// TIA Portal V17 export
// export: Created 2023-03-06T02:05:17.4655163Z, ExportSetting WithDefaults, DisplayName Totally Integrated Automation Portal, DisplayVersion V17 Update 4, DisplayName TIA Portal Openness, DisplayVersion V17 Update 4, DisplayName TIA Portal Version Control Interface, DisplayVersion V17, DisplayName STEP 7 Professional, DisplayVersion V17 Update 4, DisplayName STEP 7 Safety, DisplayVersion V17, DisplayName WinCC Professional, DisplayVersion V17 Update 4
FUNCTION "AssetSt" : Void   // FC122, LAD
{ S7_Optimized_Access := 'TRUE' }
VERSION : 0.1
// stored: AutoNumber false, IsIECCheckEnabled false, SetENOAutomatically false, UDAEnableTagReadback false
BEGIN

REGION Network 1: Asset Status Battery Bank 1
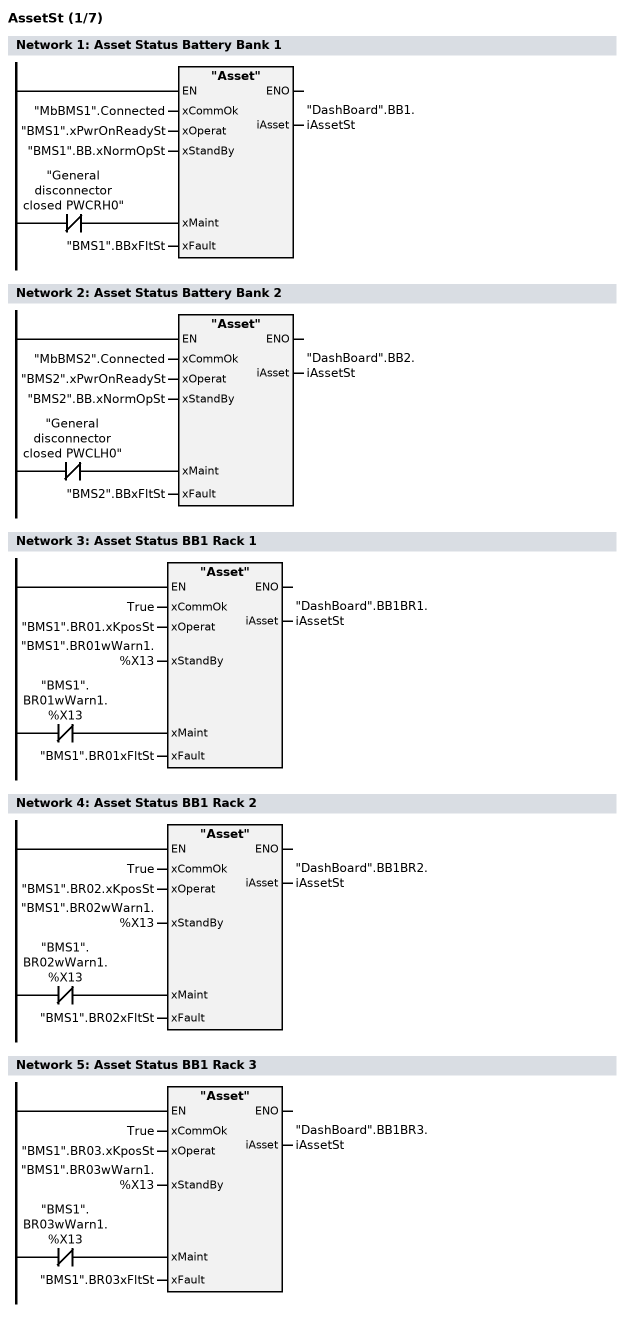
   RUNG wire#powerrail
      "Asset"(xMaint := wire#w1, xCommOk := "MbBMS1".Connected, xOperat := "BMS1".xPwrOnReadySt, xStandBy := "BMS1".BB.xNormOpSt, xFault := "BMS1".BBxFltSt, iAsset => "DashBoard".BB1.iAssetSt)
   END_RUNG
   RUNG wire#powerrail
      I_Contact( "General disconnector closed PWCRH0" )
   END_RUNG wire#w1
   // the same network as SCL:
   "Asset"(xCommOk := "MbBMS1".Connected,
           xOperat := "BMS1".xPwrOnReadySt,
           xStandBy := "BMS1".BB.xNormOpSt,
           xMaint := NOT "General disconnector closed PWCRH0",
           xFault := "BMS1".BBxFltSt,
           iAsset => "DashBoard".BB1.iAssetSt);
END_REGION

REGION Network 2: Asset Status Battery Bank 2
   RUNG wire#powerrail
      "Asset"(xMaint := wire#w1, xCommOk := "MbBMS2".Connected, xOperat := "BMS2".xPwrOnReadySt, xStandBy := "BMS2".BB.xNormOpSt, xFault := "BMS2".BBxFltSt, iAsset => "DashBoard".BB2.iAssetSt)
   END_RUNG
   RUNG wire#powerrail
      I_Contact( "General disconnector closed PWCLH0" )
   END_RUNG wire#w1
   // the same network as SCL:
   "Asset"(xCommOk := "MbBMS2".Connected,
           xOperat := "BMS2".xPwrOnReadySt,
           xStandBy := "BMS2".BB.xNormOpSt,
           xMaint := NOT "General disconnector closed PWCLH0",
           xFault := "BMS2".BBxFltSt,
           iAsset => "DashBoard".BB2.iAssetSt);
END_REGION

REGION Network 3: Asset Status BB1 Rack 1
   RUNG wire#powerrail
      "Asset"(xMaint := wire#w1, xCommOk := True, xOperat := "BMS1".BR01.xKposSt, xStandBy := "BMS1".BR01wWarn1.%X13, xFault := "BMS1".BR01xFltSt, iAsset => "DashBoard".BB1BR1.iAssetSt)
   END_RUNG
   RUNG wire#powerrail
      I_Contact( "BMS1".BR01wWarn1.%X13 )
   END_RUNG wire#w1
   // the same network as SCL:
   "Asset"(xCommOk := True,
           xOperat := "BMS1".BR01.xKposSt,
           xStandBy := "BMS1".BR01wWarn1.%X13,
           xMaint := NOT "BMS1".BR01wWarn1.%X13,
           xFault := "BMS1".BR01xFltSt,
           iAsset => "DashBoard".BB1BR1.iAssetSt);
END_REGION

REGION Network 4: Asset Status BB1 Rack 2
   RUNG wire#powerrail
      "Asset"(xMaint := wire#w1, xCommOk := True, xOperat := "BMS1".BR02.xKposSt, xStandBy := "BMS1".BR02wWarn1.%X13, xFault := "BMS1".BR02xFltSt, iAsset => "DashBoard".BB1BR2.iAssetSt)
   END_RUNG
   RUNG wire#powerrail
      I_Contact( "BMS1".BR02wWarn1.%X13 )
   END_RUNG wire#w1
   // the same network as SCL:
   "Asset"(xCommOk := True,
           xOperat := "BMS1".BR02.xKposSt,
           xStandBy := "BMS1".BR02wWarn1.%X13,
           xMaint := NOT "BMS1".BR02wWarn1.%X13,
           xFault := "BMS1".BR02xFltSt,
           iAsset => "DashBoard".BB1BR2.iAssetSt);
END_REGION

REGION Network 5: Asset Status BB1 Rack 3
   RUNG wire#powerrail
      "Asset"(xMaint := wire#w1, xCommOk := True, xOperat := "BMS1".BR03.xKposSt, xStandBy := "BMS1".BR03wWarn1.%X13, xFault := "BMS1".BR03xFltSt, iAsset => "DashBoard".BB1BR3.iAssetSt)
   END_RUNG
   RUNG wire#powerrail
      I_Contact( "BMS1".BR03wWarn1.%X13 )
   END_RUNG wire#w1
   // the same network as SCL:
   "Asset"(xCommOk := True,
           xOperat := "BMS1".BR03.xKposSt,
           xStandBy := "BMS1".BR03wWarn1.%X13,
           xMaint := NOT "BMS1".BR03wWarn1.%X13,
           xFault := "BMS1".BR03xFltSt,
           iAsset => "DashBoard".BB1BR3.iAssetSt);
END_REGION

REGION Network 6: Asset Status BB1 Rack 4
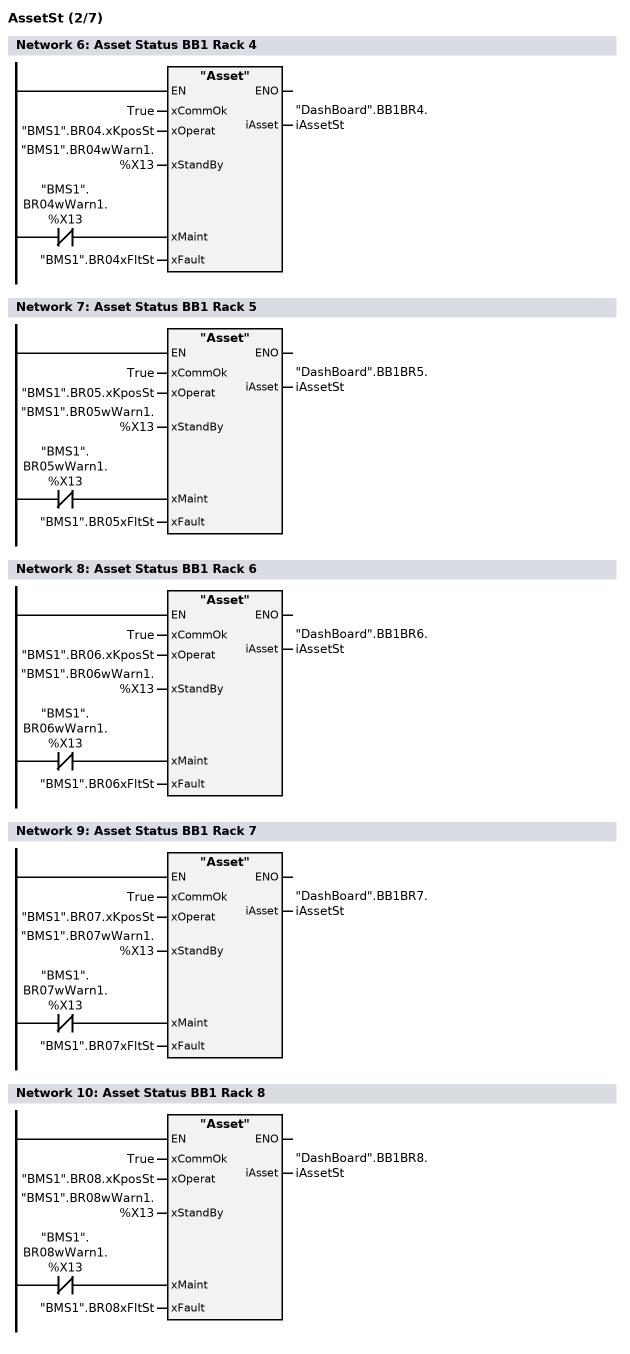
   RUNG wire#powerrail
      "Asset"(xMaint := wire#w1, xCommOk := True, xOperat := "BMS1".BR04.xKposSt, xStandBy := "BMS1".BR04wWarn1.%X13, xFault := "BMS1".BR04xFltSt, iAsset => "DashBoard".BB1BR4.iAssetSt)
   END_RUNG
   RUNG wire#powerrail
      I_Contact( "BMS1".BR04wWarn1.%X13 )
   END_RUNG wire#w1
   // the same network as SCL:
   "Asset"(xCommOk := True,
           xOperat := "BMS1".BR04.xKposSt,
           xStandBy := "BMS1".BR04wWarn1.%X13,
           xMaint := NOT "BMS1".BR04wWarn1.%X13,
           xFault := "BMS1".BR04xFltSt,
           iAsset => "DashBoard".BB1BR4.iAssetSt);
END_REGION

REGION Network 7: Asset Status BB1 Rack 5
   RUNG wire#powerrail
      "Asset"(xMaint := wire#w1, xCommOk := True, xOperat := "BMS1".BR05.xKposSt, xStandBy := "BMS1".BR05wWarn1.%X13, xFault := "BMS1".BR05xFltSt, iAsset => "DashBoard".BB1BR5.iAssetSt)
   END_RUNG
   RUNG wire#powerrail
      I_Contact( "BMS1".BR05wWarn1.%X13 )
   END_RUNG wire#w1
   // the same network as SCL:
   "Asset"(xCommOk := True,
           xOperat := "BMS1".BR05.xKposSt,
           xStandBy := "BMS1".BR05wWarn1.%X13,
           xMaint := NOT "BMS1".BR05wWarn1.%X13,
           xFault := "BMS1".BR05xFltSt,
           iAsset => "DashBoard".BB1BR5.iAssetSt);
END_REGION

REGION Network 8: Asset Status BB1 Rack 6
   RUNG wire#powerrail
      "Asset"(xMaint := wire#w1, xCommOk := True, xOperat := "BMS1".BR06.xKposSt, xStandBy := "BMS1".BR06wWarn1.%X13, xFault := "BMS1".BR06xFltSt, iAsset => "DashBoard".BB1BR6.iAssetSt)
   END_RUNG
   RUNG wire#powerrail
      I_Contact( "BMS1".BR06wWarn1.%X13 )
   END_RUNG wire#w1
   // the same network as SCL:
   "Asset"(xCommOk := True,
           xOperat := "BMS1".BR06.xKposSt,
           xStandBy := "BMS1".BR06wWarn1.%X13,
           xMaint := NOT "BMS1".BR06wWarn1.%X13,
           xFault := "BMS1".BR06xFltSt,
           iAsset => "DashBoard".BB1BR6.iAssetSt);
END_REGION

REGION Network 9: Asset Status BB1 Rack 7
   RUNG wire#powerrail
      "Asset"(xMaint := wire#w1, xCommOk := True, xOperat := "BMS1".BR07.xKposSt, xStandBy := "BMS1".BR07wWarn1.%X13, xFault := "BMS1".BR07xFltSt, iAsset => "DashBoard".BB1BR7.iAssetSt)
   END_RUNG
   RUNG wire#powerrail
      I_Contact( "BMS1".BR07wWarn1.%X13 )
   END_RUNG wire#w1
   // the same network as SCL:
   "Asset"(xCommOk := True,
           xOperat := "BMS1".BR07.xKposSt,
           xStandBy := "BMS1".BR07wWarn1.%X13,
           xMaint := NOT "BMS1".BR07wWarn1.%X13,
           xFault := "BMS1".BR07xFltSt,
           iAsset => "DashBoard".BB1BR7.iAssetSt);
END_REGION

REGION Network 10: Asset Status BB1 Rack 8
   RUNG wire#powerrail
      "Asset"(xMaint := wire#w1, xCommOk := True, xOperat := "BMS1".BR08.xKposSt, xStandBy := "BMS1".BR08wWarn1.%X13, xFault := "BMS1".BR08xFltSt, iAsset => "DashBoard".BB1BR8.iAssetSt)
   END_RUNG
   RUNG wire#powerrail
      I_Contact( "BMS1".BR08wWarn1.%X13 )
   END_RUNG wire#w1
   // the same network as SCL:
   "Asset"(xCommOk := True,
           xOperat := "BMS1".BR08.xKposSt,
           xStandBy := "BMS1".BR08wWarn1.%X13,
           xMaint := NOT "BMS1".BR08wWarn1.%X13,
           xFault := "BMS1".BR08xFltSt,
           iAsset => "DashBoard".BB1BR8.iAssetSt);
END_REGION

REGION Network 11: Asset Status BB1 Rack 9
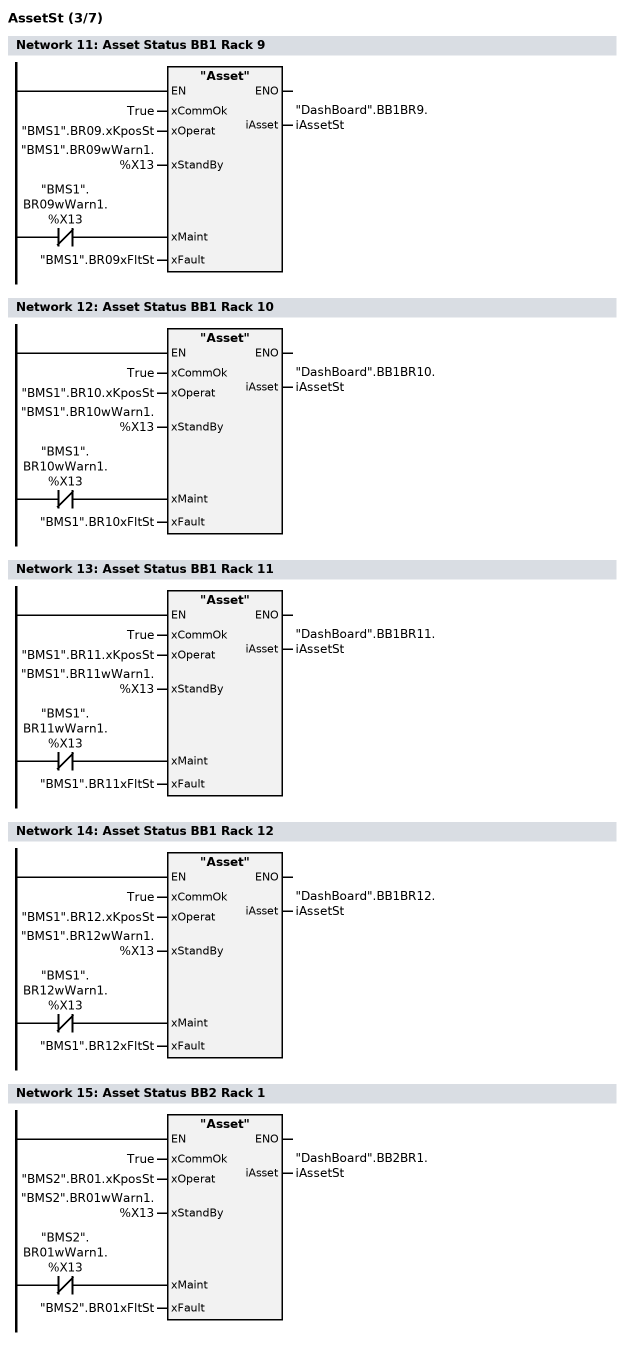
   RUNG wire#powerrail
      "Asset"(xMaint := wire#w1, xCommOk := True, xOperat := "BMS1".BR09.xKposSt, xStandBy := "BMS1".BR09wWarn1.%X13, xFault := "BMS1".BR09xFltSt, iAsset => "DashBoard".BB1BR9.iAssetSt)
   END_RUNG
   RUNG wire#powerrail
      I_Contact( "BMS1".BR09wWarn1.%X13 )
   END_RUNG wire#w1
   // the same network as SCL:
   "Asset"(xCommOk := True,
           xOperat := "BMS1".BR09.xKposSt,
           xStandBy := "BMS1".BR09wWarn1.%X13,
           xMaint := NOT "BMS1".BR09wWarn1.%X13,
           xFault := "BMS1".BR09xFltSt,
           iAsset => "DashBoard".BB1BR9.iAssetSt);
END_REGION

REGION Network 12: Asset Status BB1 Rack 10
   RUNG wire#powerrail
      "Asset"(xMaint := wire#w1, xCommOk := True, xOperat := "BMS1".BR10.xKposSt, xStandBy := "BMS1".BR10wWarn1.%X13, xFault := "BMS1".BR10xFltSt, iAsset => "DashBoard".BB1BR10.iAssetSt)
   END_RUNG
   RUNG wire#powerrail
      I_Contact( "BMS1".BR10wWarn1.%X13 )
   END_RUNG wire#w1
   // the same network as SCL:
   "Asset"(xCommOk := True,
           xOperat := "BMS1".BR10.xKposSt,
           xStandBy := "BMS1".BR10wWarn1.%X13,
           xMaint := NOT "BMS1".BR10wWarn1.%X13,
           xFault := "BMS1".BR10xFltSt,
           iAsset => "DashBoard".BB1BR10.iAssetSt);
END_REGION

REGION Network 13: Asset Status BB1 Rack 11
   RUNG wire#powerrail
      "Asset"(xMaint := wire#w1, xCommOk := True, xOperat := "BMS1".BR11.xKposSt, xStandBy := "BMS1".BR11wWarn1.%X13, xFault := "BMS1".BR11xFltSt, iAsset => "DashBoard".BB1BR11.iAssetSt)
   END_RUNG
   RUNG wire#powerrail
      I_Contact( "BMS1".BR11wWarn1.%X13 )
   END_RUNG wire#w1
   // the same network as SCL:
   "Asset"(xCommOk := True,
           xOperat := "BMS1".BR11.xKposSt,
           xStandBy := "BMS1".BR11wWarn1.%X13,
           xMaint := NOT "BMS1".BR11wWarn1.%X13,
           xFault := "BMS1".BR11xFltSt,
           iAsset => "DashBoard".BB1BR11.iAssetSt);
END_REGION

REGION Network 14: Asset Status BB1 Rack 12
   RUNG wire#powerrail
      "Asset"(xMaint := wire#w1, xCommOk := True, xOperat := "BMS1".BR12.xKposSt, xStandBy := "BMS1".BR12wWarn1.%X13, xFault := "BMS1".BR12xFltSt, iAsset => "DashBoard".BB1BR12.iAssetSt)
   END_RUNG
   RUNG wire#powerrail
      I_Contact( "BMS1".BR12wWarn1.%X13 )
   END_RUNG wire#w1
   // the same network as SCL:
   "Asset"(xCommOk := True,
           xOperat := "BMS1".BR12.xKposSt,
           xStandBy := "BMS1".BR12wWarn1.%X13,
           xMaint := NOT "BMS1".BR12wWarn1.%X13,
           xFault := "BMS1".BR12xFltSt,
           iAsset => "DashBoard".BB1BR12.iAssetSt);
END_REGION

REGION Network 15: Asset Status BB2 Rack 1
   RUNG wire#powerrail
      "Asset"(xMaint := wire#w1, xCommOk := True, xOperat := "BMS2".BR01.xKposSt, xStandBy := "BMS2".BR01wWarn1.%X13, xFault := "BMS2".BR01xFltSt, iAsset => "DashBoard".BB2BR1.iAssetSt)
   END_RUNG
   RUNG wire#powerrail
      I_Contact( "BMS2".BR01wWarn1.%X13 )
   END_RUNG wire#w1
   // the same network as SCL:
   "Asset"(xCommOk := True,
           xOperat := "BMS2".BR01.xKposSt,
           xStandBy := "BMS2".BR01wWarn1.%X13,
           xMaint := NOT "BMS2".BR01wWarn1.%X13,
           xFault := "BMS2".BR01xFltSt,
           iAsset => "DashBoard".BB2BR1.iAssetSt);
END_REGION

REGION Network 16: Asset Status BB2 Rack 2
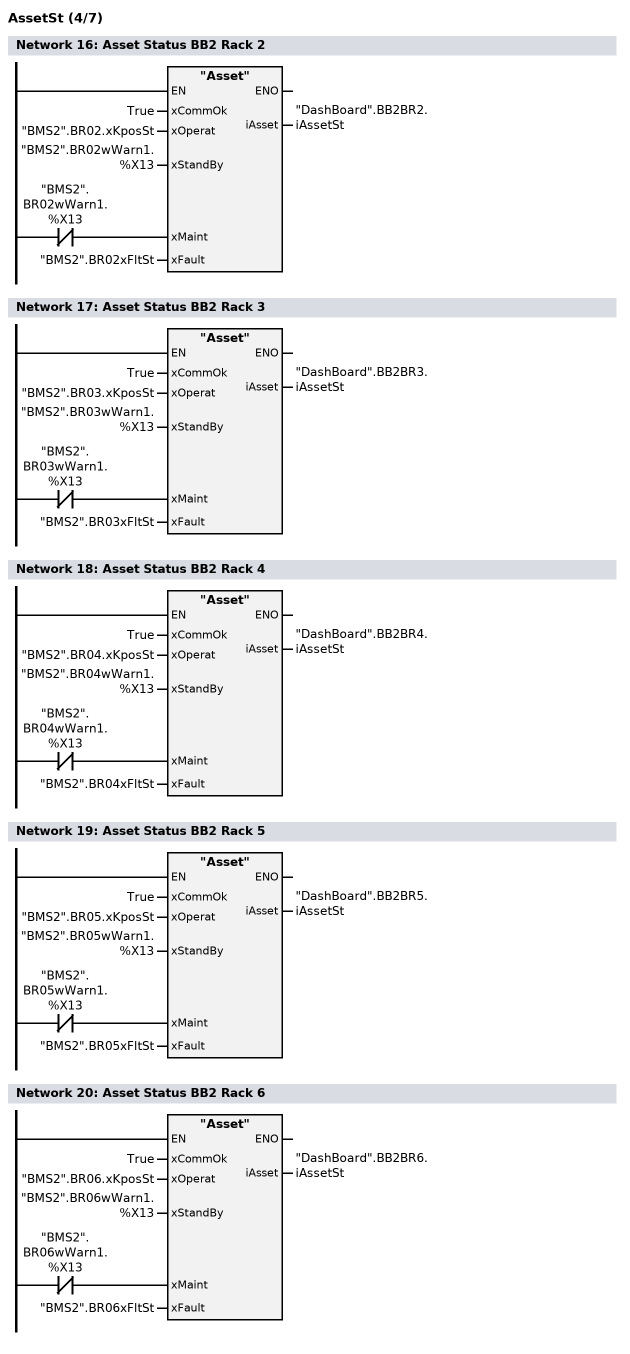
   RUNG wire#powerrail
      "Asset"(xMaint := wire#w1, xCommOk := True, xOperat := "BMS2".BR02.xKposSt, xStandBy := "BMS2".BR02wWarn1.%X13, xFault := "BMS2".BR02xFltSt, iAsset => "DashBoard".BB2BR2.iAssetSt)
   END_RUNG
   RUNG wire#powerrail
      I_Contact( "BMS2".BR02wWarn1.%X13 )
   END_RUNG wire#w1
   // the same network as SCL:
   "Asset"(xCommOk := True,
           xOperat := "BMS2".BR02.xKposSt,
           xStandBy := "BMS2".BR02wWarn1.%X13,
           xMaint := NOT "BMS2".BR02wWarn1.%X13,
           xFault := "BMS2".BR02xFltSt,
           iAsset => "DashBoard".BB2BR2.iAssetSt);
END_REGION

REGION Network 17: Asset Status BB2 Rack 3
   RUNG wire#powerrail
      "Asset"(xMaint := wire#w1, xCommOk := True, xOperat := "BMS2".BR03.xKposSt, xStandBy := "BMS2".BR03wWarn1.%X13, xFault := "BMS2".BR03xFltSt, iAsset => "DashBoard".BB2BR3.iAssetSt)
   END_RUNG
   RUNG wire#powerrail
      I_Contact( "BMS2".BR03wWarn1.%X13 )
   END_RUNG wire#w1
   // the same network as SCL:
   "Asset"(xCommOk := True,
           xOperat := "BMS2".BR03.xKposSt,
           xStandBy := "BMS2".BR03wWarn1.%X13,
           xMaint := NOT "BMS2".BR03wWarn1.%X13,
           xFault := "BMS2".BR03xFltSt,
           iAsset => "DashBoard".BB2BR3.iAssetSt);
END_REGION

REGION Network 18: Asset Status BB2 Rack 4
   RUNG wire#powerrail
      "Asset"(xMaint := wire#w1, xCommOk := True, xOperat := "BMS2".BR04.xKposSt, xStandBy := "BMS2".BR04wWarn1.%X13, xFault := "BMS2".BR04xFltSt, iAsset => "DashBoard".BB2BR4.iAssetSt)
   END_RUNG
   RUNG wire#powerrail
      I_Contact( "BMS2".BR04wWarn1.%X13 )
   END_RUNG wire#w1
   // the same network as SCL:
   "Asset"(xCommOk := True,
           xOperat := "BMS2".BR04.xKposSt,
           xStandBy := "BMS2".BR04wWarn1.%X13,
           xMaint := NOT "BMS2".BR04wWarn1.%X13,
           xFault := "BMS2".BR04xFltSt,
           iAsset => "DashBoard".BB2BR4.iAssetSt);
END_REGION

REGION Network 19: Asset Status BB2 Rack 5
   RUNG wire#powerrail
      "Asset"(xMaint := wire#w1, xCommOk := True, xOperat := "BMS2".BR05.xKposSt, xStandBy := "BMS2".BR05wWarn1.%X13, xFault := "BMS2".BR05xFltSt, iAsset => "DashBoard".BB2BR5.iAssetSt)
   END_RUNG
   RUNG wire#powerrail
      I_Contact( "BMS2".BR05wWarn1.%X13 )
   END_RUNG wire#w1
   // the same network as SCL:
   "Asset"(xCommOk := True,
           xOperat := "BMS2".BR05.xKposSt,
           xStandBy := "BMS2".BR05wWarn1.%X13,
           xMaint := NOT "BMS2".BR05wWarn1.%X13,
           xFault := "BMS2".BR05xFltSt,
           iAsset => "DashBoard".BB2BR5.iAssetSt);
END_REGION

REGION Network 20: Asset Status BB2 Rack 6
   RUNG wire#powerrail
      "Asset"(xMaint := wire#w1, xCommOk := True, xOperat := "BMS2".BR06.xKposSt, xStandBy := "BMS2".BR06wWarn1.%X13, xFault := "BMS2".BR06xFltSt, iAsset => "DashBoard".BB2BR6.iAssetSt)
   END_RUNG
   RUNG wire#powerrail
      I_Contact( "BMS2".BR06wWarn1.%X13 )
   END_RUNG wire#w1
   // the same network as SCL:
   "Asset"(xCommOk := True,
           xOperat := "BMS2".BR06.xKposSt,
           xStandBy := "BMS2".BR06wWarn1.%X13,
           xMaint := NOT "BMS2".BR06wWarn1.%X13,
           xFault := "BMS2".BR06xFltSt,
           iAsset => "DashBoard".BB2BR6.iAssetSt);
END_REGION

REGION Network 21: Asset Status BB2 Rack 7
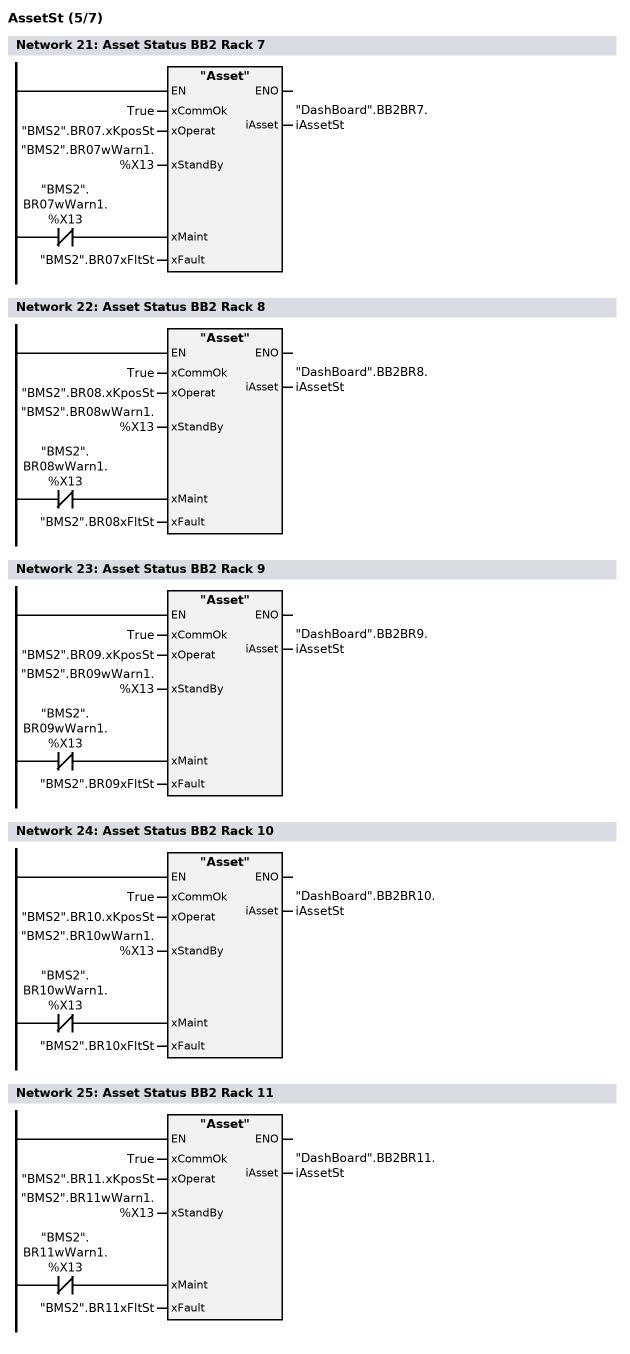
   RUNG wire#powerrail
      "Asset"(xMaint := wire#w1, xCommOk := True, xOperat := "BMS2".BR07.xKposSt, xStandBy := "BMS2".BR07wWarn1.%X13, xFault := "BMS2".BR07xFltSt, iAsset => "DashBoard".BB2BR7.iAssetSt)
   END_RUNG
   RUNG wire#powerrail
      I_Contact( "BMS2".BR07wWarn1.%X13 )
   END_RUNG wire#w1
   // the same network as SCL:
   "Asset"(xCommOk := True,
           xOperat := "BMS2".BR07.xKposSt,
           xStandBy := "BMS2".BR07wWarn1.%X13,
           xMaint := NOT "BMS2".BR07wWarn1.%X13,
           xFault := "BMS2".BR07xFltSt,
           iAsset => "DashBoard".BB2BR7.iAssetSt);
END_REGION

REGION Network 22: Asset Status BB2 Rack 8
   RUNG wire#powerrail
      "Asset"(xMaint := wire#w1, xCommOk := True, xOperat := "BMS2".BR08.xKposSt, xStandBy := "BMS2".BR08wWarn1.%X13, xFault := "BMS2".BR08xFltSt, iAsset => "DashBoard".BB2BR8.iAssetSt)
   END_RUNG
   RUNG wire#powerrail
      I_Contact( "BMS2".BR08wWarn1.%X13 )
   END_RUNG wire#w1
   // the same network as SCL:
   "Asset"(xCommOk := True,
           xOperat := "BMS2".BR08.xKposSt,
           xStandBy := "BMS2".BR08wWarn1.%X13,
           xMaint := NOT "BMS2".BR08wWarn1.%X13,
           xFault := "BMS2".BR08xFltSt,
           iAsset => "DashBoard".BB2BR8.iAssetSt);
END_REGION

REGION Network 23: Asset Status BB2 Rack 9
   RUNG wire#powerrail
      "Asset"(xMaint := wire#w1, xCommOk := True, xOperat := "BMS2".BR09.xKposSt, xStandBy := "BMS2".BR09wWarn1.%X13, xFault := "BMS2".BR09xFltSt, iAsset => "DashBoard".BB2BR9.iAssetSt)
   END_RUNG
   RUNG wire#powerrail
      I_Contact( "BMS2".BR09wWarn1.%X13 )
   END_RUNG wire#w1
   // the same network as SCL:
   "Asset"(xCommOk := True,
           xOperat := "BMS2".BR09.xKposSt,
           xStandBy := "BMS2".BR09wWarn1.%X13,
           xMaint := NOT "BMS2".BR09wWarn1.%X13,
           xFault := "BMS2".BR09xFltSt,
           iAsset => "DashBoard".BB2BR9.iAssetSt);
END_REGION

REGION Network 24: Asset Status BB2 Rack 10
   RUNG wire#powerrail
      "Asset"(xMaint := wire#w1, xCommOk := True, xOperat := "BMS2".BR10.xKposSt, xStandBy := "BMS2".BR10wWarn1.%X13, xFault := "BMS2".BR10xFltSt, iAsset => "DashBoard".BB2BR10.iAssetSt)
   END_RUNG
   RUNG wire#powerrail
      I_Contact( "BMS2".BR10wWarn1.%X13 )
   END_RUNG wire#w1
   // the same network as SCL:
   "Asset"(xCommOk := True,
           xOperat := "BMS2".BR10.xKposSt,
           xStandBy := "BMS2".BR10wWarn1.%X13,
           xMaint := NOT "BMS2".BR10wWarn1.%X13,
           xFault := "BMS2".BR10xFltSt,
           iAsset => "DashBoard".BB2BR10.iAssetSt);
END_REGION

REGION Network 25: Asset Status BB2 Rack 11
   RUNG wire#powerrail
      "Asset"(xMaint := wire#w1, xCommOk := True, xOperat := "BMS2".BR11.xKposSt, xStandBy := "BMS2".BR11wWarn1.%X13, xFault := "BMS2".BR11xFltSt, iAsset => "DashBoard".BB2BR11.iAssetSt)
   END_RUNG
   RUNG wire#powerrail
      I_Contact( "BMS2".BR11wWarn1.%X13 )
   END_RUNG wire#w1
   // the same network as SCL:
   "Asset"(xCommOk := True,
           xOperat := "BMS2".BR11.xKposSt,
           xStandBy := "BMS2".BR11wWarn1.%X13,
           xMaint := NOT "BMS2".BR11wWarn1.%X13,
           xFault := "BMS2".BR11xFltSt,
           iAsset => "DashBoard".BB2BR11.iAssetSt);
END_REGION

REGION Network 26: Asset Status BB2 Rack 12
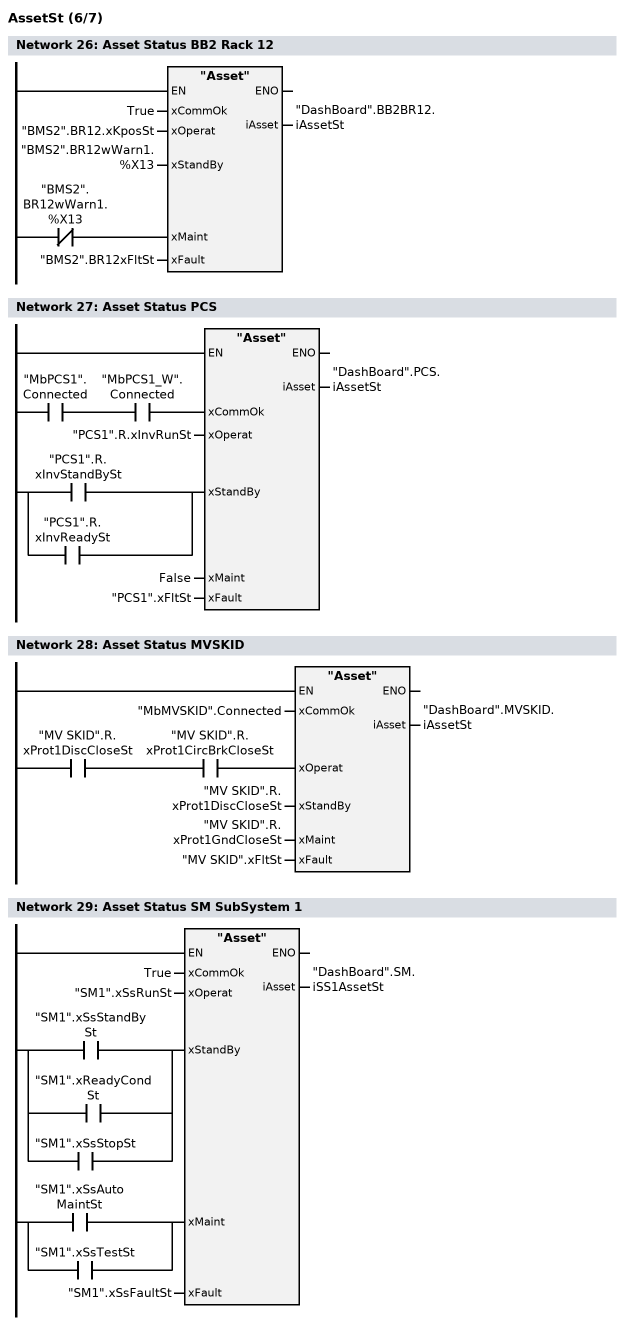
   RUNG wire#powerrail
      "Asset"(xMaint := wire#w1, xCommOk := True, xOperat := "BMS2".BR12.xKposSt, xStandBy := "BMS2".BR12wWarn1.%X13, xFault := "BMS2".BR12xFltSt, iAsset => "DashBoard".BB2BR12.iAssetSt)
   END_RUNG
   RUNG wire#powerrail
      I_Contact( "BMS2".BR12wWarn1.%X13 )
   END_RUNG wire#w1
   // the same network as SCL:
   "Asset"(xCommOk := True,
           xOperat := "BMS2".BR12.xKposSt,
           xStandBy := "BMS2".BR12wWarn1.%X13,
           xMaint := NOT "BMS2".BR12wWarn1.%X13,
           xFault := "BMS2".BR12xFltSt,
           iAsset => "DashBoard".BB2BR12.iAssetSt);
END_REGION

REGION Network 27: Asset Status PCS
   RUNG wire#powerrail
      "Asset"(xCommOk := wire#w1, xStandBy := wire#w2, xOperat := "PCS1".R.xInvRunSt, xMaint := False, xFault := "PCS1".xFltSt, iAsset => "DashBoard".PCS.iAssetSt)
   END_RUNG
   RUNG wire#powerrail
      Contact( "MbPCS1".Connected )
      Contact( "MbPCS1_W".Connected )
   END_RUNG wire#w1
   RUNG wire#powerrail
      Contact( "PCS1".R.xInvStandBySt )
   END_RUNG wire#w2
   RUNG wire#powerrail
      Contact( "PCS1".R.xInvReadySt )
   END_RUNG wire#w2
   // the same network as SCL:
   "Asset"(xCommOk := "MbPCS1".Connected AND "MbPCS1_W".Connected,
           xOperat := "PCS1".R.xInvRunSt,
           xStandBy := "PCS1".R.xInvStandBySt OR "PCS1".R.xInvReadySt,
           xMaint := False,
           xFault := "PCS1".xFltSt,
           iAsset => "DashBoard".PCS.iAssetSt);
END_REGION

REGION Network 28: Asset Status MVSKID
   RUNG wire#powerrail
      "Asset"(xOperat := wire#w1, xCommOk := "MbMVSKID".Connected, xStandBy := "MV SKID".R.xProt1DiscCloseSt, xMaint := "MV SKID".R.xProt1GndCloseSt, xFault := "MV SKID".xFltSt, iAsset => "DashBoard".MVSKID.iAssetSt)
   END_RUNG
   RUNG wire#powerrail
      Contact( "MV SKID".R.xProt1DiscCloseSt )
      Contact( "MV SKID".R.xProt1CircBrkCloseSt )
   END_RUNG wire#w1
   // the same network as SCL:
   "Asset"(xCommOk := "MbMVSKID".Connected,
           xOperat := "MV SKID".R.xProt1DiscCloseSt AND "MV SKID".R.xProt1CircBrkCloseSt,
           xStandBy := "MV SKID".R.xProt1DiscCloseSt,
           xMaint := "MV SKID".R.xProt1GndCloseSt,
           xFault := "MV SKID".xFltSt,
           iAsset => "DashBoard".MVSKID.iAssetSt);
END_REGION

REGION Network 29: Asset Status SM SubSystem 1
   RUNG wire#powerrail
      "Asset"(xStandBy := wire#w1, xMaint := wire#w2, xCommOk := True, xOperat := "SM1".xSsRunSt, xFault := "SM1".xSsFaultSt, iAsset => "DashBoard".SM.iSS1AssetSt)
   END_RUNG
   RUNG wire#powerrail
      Contact( "SM1".xSsStandBySt )
   END_RUNG wire#w1
   RUNG wire#powerrail
      Contact( "SM1".xReadyCondSt )
   END_RUNG wire#w1
   RUNG wire#powerrail
      Contact( "SM1".xSsStopSt )
   END_RUNG wire#w1
   RUNG wire#powerrail
      Contact( "SM1".xSsAutoMaintSt )
   END_RUNG wire#w2
   RUNG wire#powerrail
      Contact( "SM1".xSsTestSt )
   END_RUNG wire#w2
   // the same network as SCL:
   "Asset"(xCommOk := True,
           xOperat := "SM1".xSsRunSt,
           xStandBy := "SM1".xSsStandBySt OR "SM1".xReadyCondSt OR "SM1".xSsStopSt,
           xMaint := "SM1".xSsAutoMaintSt OR "SM1".xSsTestSt,
           xFault := "SM1".xSsFaultSt,
           iAsset => "DashBoard".SM.iSS1AssetSt);
END_REGION

REGION Network 30: Asset Status SM SubSystem 2
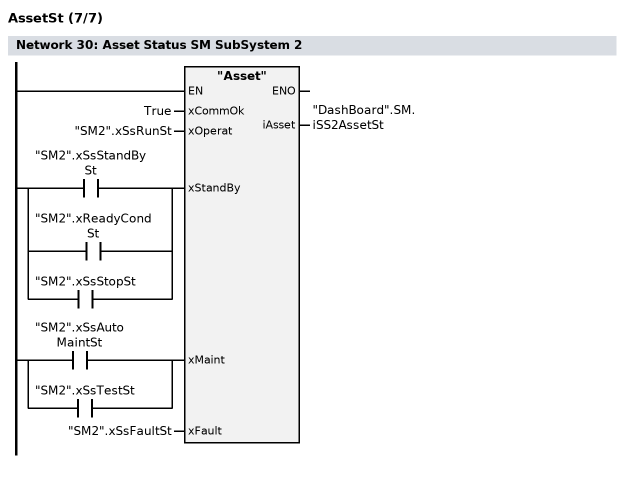
   RUNG wire#powerrail
      "Asset"(xStandBy := wire#w1, xMaint := wire#w2, xCommOk := True, xOperat := "SM2".xSsRunSt, xFault := "SM2".xSsFaultSt, iAsset => "DashBoard".SM.iSS2AssetSt)
   END_RUNG
   RUNG wire#powerrail
      Contact( "SM2".xSsStandBySt )
   END_RUNG wire#w1
   RUNG wire#powerrail
      Contact( "SM2".xReadyCondSt )
   END_RUNG wire#w1
   RUNG wire#powerrail
      Contact( "SM2".xSsStopSt )
   END_RUNG wire#w1
   RUNG wire#powerrail
      Contact( "SM2".xSsAutoMaintSt )
   END_RUNG wire#w2
   RUNG wire#powerrail
      Contact( "SM2".xSsTestSt )
   END_RUNG wire#w2
   // the same network as SCL:
   "Asset"(xCommOk := True,
           xOperat := "SM2".xSsRunSt,
           xStandBy := "SM2".xSsStandBySt OR "SM2".xReadyCondSt OR "SM2".xSsStopSt,
           xMaint := "SM2".xSsAutoMaintSt OR "SM2".xSsTestSt,
           xFault := "SM2".xSsFaultSt,
           iAsset => "DashBoard".SM.iSS2AssetSt);
END_REGION
END_FUNCTION
